{attribute 'qualified_only'}
{attribute 'strict'}
TYPE E_LED_Errors :
(
	disconnected := 0,
	none := 1
);
END_TYPE

(* stored: Version 1.1.0.1, ProductVersion 3.1.4022.12
   DUT E_LED_Errors: Id {bc3bcf87-60b6-4ef0-91c7-c25055c3333e} *)
